// TIA Portal V18 export
DATA_BLOCK "HeatingPLC_vDO_Vars"   // DB11004
{ S7_Optimized_Access := 'FALSE' }
VERSION : 0.1
// stored: AutoNumber false, DBAccessibleFromOPCUA true, IsOnlyStoredInLoadMemory false, IsWriteProtectedInAS false
   VAR
      vDO1 { S7_SetPoint := 'True'} : "UDT_vDO";
      vDO2 { S7_SetPoint := 'True'} : "UDT_vDO";
      vDO3 { S7_SetPoint := 'True'} : "UDT_vDO";
      vDO4 { S7_SetPoint := 'True'} : "UDT_vDO";
      vDO5 { S7_SetPoint := 'True'} : "UDT_vDO";
      vDO6 { S7_SetPoint := 'True'} : "UDT_vDO";
      vDO7 { S7_SetPoint := 'True'} : "UDT_vDO";
      vDO8 { S7_SetPoint := 'True'} : "UDT_vDO";
   END_VAR
BEGIN
END_DATA_BLOCK
